Fanuc KAREL source: APPEND_QUEUE.kl

PROGRAM T
%NOLOCKGROUP
VAR
 v0 : INTEGER
 v1 : QUEUE_TYPE
 v2 : ARRAY[10] OF INTEGER
 v3 : INTEGER
 v4 : INTEGER
BEGIN
 APPEND_QUEUE(v0, v1, v2, v3, v4)
END T
